{attribute 'linkalways'} 
{attribute 'no_explicit_call' := 'This FB is a CLASS and must be accessed using methods or properties'}
{attribute 'enable_dynamic_creation'}
FUNCTION_BLOCK ABSTRACT DatatypeBase EXTENDS Disposable IMPLEMENTS I_Datatype
VAR
END_VAR

METHOD PUBLIC Accept
VAR_INPUT
	Visitor : I_DatatypeVisitor;
END_VAR
Visitor.VisitDatatype(this^);
END_METHOD

PROPERTY PUBLIC ABSTRACT Address : PVOID
GET
END_GET
END_PROPERTY

METHOD PUBLIC ABSTRACT ClearReference
VAR_INPUT
END_VAR
END_METHOD

METHOD PUBLIC ABSTRACT Clone : I_Datatype
END_METHOD

PROPERTY PUBLIC IsUserDefined : BOOL
GET
IsUserDefined := FALSE;
END_GET
END_PROPERTY

METHOD PROTECTED OnSerializeTypeWith
VAR_INPUT
	Serializer : I_Serializer;
END_VAR
Serializer.AddKeyString('typeName',TypeName);
END_METHOD

METHOD PUBLIC SerializeTypeWith
VAR_INPUT
	Serializer : I_Serializer;
END_VAR
Serializer.StartObject();
OnSerializeTypeWith(Serializer);
Serializer.EndObject();
END_METHOD

METHOD PUBLIC ABSTRACT SerializeWith
VAR_INPUT
	Serializer : I_Serializer;
END_VAR
END_METHOD

PROPERTY PUBLIC ABSTRACT Size : UDINT
GET
END_GET
END_PROPERTY

METHOD PUBLIC TryCopyFrom : BOOL
VAR_INPUT
	Source : I_Datatype;
END_VAR
IF Source.TypeName <> TypeName THEN
	RETURN;
END_IF

memcpy(Address, Source.Address, Size);
TryCopyFrom := TRUE;
END_METHOD

METHOD PUBLIC ABSTRACT TryDeserializeFrom : BOOL
VAR_INPUT
	Deserializer : I_Deserializer;
	Feedback : I_DeserializerFeedback;
END_VAR
END_METHOD

METHOD PUBLIC ABSTRACT TryMakeReferenceTo : BOOL
VAR_INPUT
	Target : I_Datatype;
END_VAR
END_METHOD

METHOD PUBLIC TryResolveAsAliasDatatype : BOOL
VAR_INPUT
	Destination : REFERENCE TO I_AliasDatatype;
END_VAR
TryResolveAsAliasDatatype := FALSE;
END_METHOD

METHOD PUBLIC TryResolveAsBitDatatype : BOOL
VAR_INPUT
	Destination : REFERENCE TO I_BitDatatype;
END_VAR
TryResolveAsBitDatatype := FALSE;
END_METHOD

METHOD PUBLIC TryResolveAsEnumDatatype : BOOL
VAR_INPUT
	Destination : REFERENCE TO I_EnumDatatype;
END_VAR
TryResolveAsEnumDatatype := FALSE;
END_METHOD

METHOD PUBLIC TryResolveAsInterfaceDatatype : BOOL
VAR_INPUT
	Destination : REFERENCE TO I_InterfaceDatatype;
END_VAR
TryResolveAsInterfaceDatatype := FALSE;
END_METHOD

METHOD PUBLIC TryResolveAsStructuredDatatype : BOOL
VAR_INPUT
	Destination : REFERENCE TO I_StructuredDatatype;
END_VAR
TryResolveAsStructuredDatatype := FALSE;
END_METHOD

PROPERTY PUBLIC ABSTRACT TypeName : T_MAXSTRING
GET
END_GET
END_PROPERTY

END_FUNCTION_BLOCK

(* stored: Version 1.1.0.1, ProductVersion 3.1.4024.12
   POU DatatypeBase: Id {f1308857-8bde-075c-0685-2da651a42b2c}, SpecialFunc None
   Folder Protected: Id {48b6bb47-c276-00f0-25e0-4934e60ec871}
   Method Accept: Id {3c6d046e-c0ee-05c3-14c2-b096a9e47227}
   Property Address: Id {8a940ee1-25f7-0552-27b0-4e429f952fd8}
   Get Get: Id {8b3ea5ed-0ab1-06f6-0b31-93fbb0622352}
   Method ClearReference: Id {1af736bc-beb8-02af-0a9a-f4544c32140a}
   Method Clone: Id {e6fa2a12-8c1f-0ef1-2f34-980e633f3468}
   Property IsUserDefined: Id {8c5b0b06-69cc-4b20-ad40-040443b3a8a5}
   Get Get: Id {be3b14b1-28de-4597-929b-49bb88cea57b}
   Method OnSerializeTypeWith: Id {f1402a76-5940-0dd1-07c6-3fa768a99025}
   Method SerializeTypeWith: Id {f3547df7-fbc8-0b47-3331-647f4354d06e}
   Method SerializeWith: Id {bacd8133-13ae-048a-1079-c7aa02210882}
   Property Size: Id {a595244c-6224-02df-3819-999db1dc5fa1}
   Get Get: Id {ea5e0ea5-6e87-0cbe-20c0-75eaad770e05}
   Method TryCopyFrom: Id {dda7c095-b8c6-0f87-2d33-9c86847656e6}
   Method TryDeserializeFrom: Id {6ff66c89-37a6-0a85-2c7a-e98c41f8fe79}
   Method TryMakeReferenceTo: Id {2f0071b8-9ed5-09d0-0263-1ad9cb921129}
   Method TryResolveAsAliasDatatype: Id {bb16e986-ad00-0935-3700-802a7bf0a865}
   Method TryResolveAsBitDatatype: Id {808046e5-2e02-482b-a556-e5322d066789}
   Method TryResolveAsEnumDatatype: Id {230d8c4f-22b2-0f35-3926-1b98347fe0f3}
   Method TryResolveAsInterfaceDatatype: Id {6cf02555-10e8-479d-a01c-2d8ef7a87819}
   Method TryResolveAsStructuredDatatype: Id {8414d3d0-ab49-0376-0d4e-3e1a2192f4ac}
   Property TypeName: Id {01acfbde-fc19-0891-0625-93e10e4849b9}
   Get Get: Id {5b9e95d4-d14d-0aad-1d4b-93d8eeae9cf7} *)
